Yaskawa INFORM job: plata_tarpez_cylinder_program.JBI

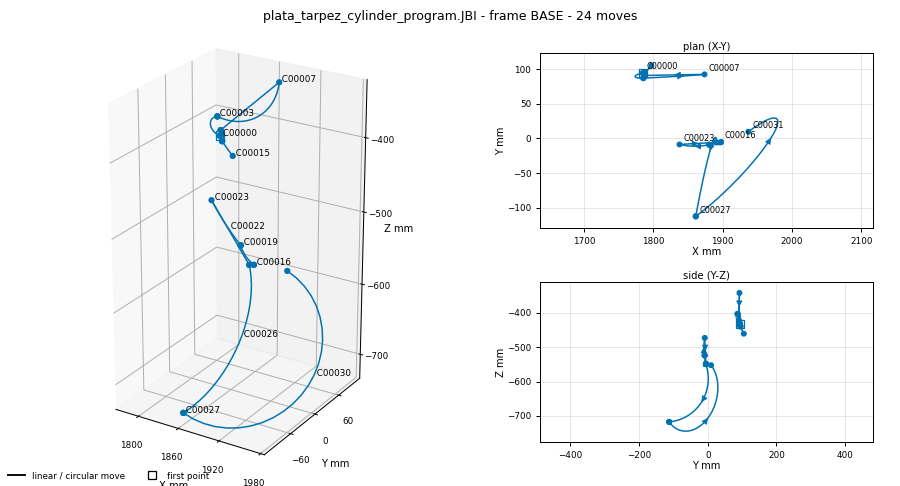
[picture p0: tool path of plata_tarpez_cylinder_program.JBI in frame BASE, 24 of 38 moves have a stored position in this frame; points joined in program order, loops and branches not executed]
/JOB
//NAME plata_tarpez_cylinder_program
//POS
///NPOS 32,0,32,0,0,0
///TOOL 0
///POSTYPE BASE
///RECTAN
///RCONF 0,0,0,0,0,0,0,0,0,0,0,0,0,0,0,0,0,0,0,0,0,0,0,0
C00000=1784.767004,94.191675,-431.505458,180.000000,-60.000000,6.127864
C00001=1784.767004,94.191675,-431.505458,180.000000,-60.000000,6.127864
C00002=1775.039434,88.021413,-411.039409,180.000000,-60.000000,7.554006
C00003=1785.526009,87.008169,-402.654234,-180.000000,-60.000000,8.255900
C00004=1785.526009,87.008169,-402.654234,-180.000000,-60.000000,8.255900
C00005=1785.526009,87.008169,-402.654234,-180.000000,-60.000000,8.255900
C00006=1813.588440,88.471809,-404.399549,-175.000000,-59.181249,9.143782
C00007=1873.697625,92.428351,-341.583881,175.000000,-33.351655,12.175617
C00008=1787.946995,90.909642,-422.120609,180.000000,-60.000000,6.802920
C00009=1787.946995,90.909642,-422.120609,180.000000,-60.000000,6.802920
C00010=1790.431356,93.825373,-431.135519,-180.000000,-60.000000,6.013660
C00011=1787.391263,95.251441,-438.765944,180.000000,-60.000000,5.494577
C00012=1787.391263,95.251441,-438.765944,180.000000,-60.000000,5.494577
C00013=1787.391263,95.251441,-438.765944,180.000000,-60.000000,5.494577
C00014=1790.708780,98.087857,-445.800605,-180.000000,-60.000000,4.731475
C00015=1797.176815,105.209463,-460.353029,180.000000,-60.000000,2.655850
C00016=1897.583937,-5.230695,-547.479957,180.000000,-60.000000,16.298157
C00017=1897.583937,-5.230695,-547.479957,180.000000,-60.000000,16.298157
C00018=1887.311406,-7.786471,-537.332214,-180.000000,-60.000000,15.451438
C00019=1880.512117,-8.938610,-523.580221,180.000000,-60.000000,14.334171
C00020=1880.512117,-8.938610,-523.580221,180.000000,-60.000000,14.334171
C00021=1880.512117,-8.938610,-523.580221,180.000000,-60.000000,14.334171
C00022=1863.998597,-11.006323,-503.995770,180.000000,-60.000000,12.058204
C00023=1837.651613,-8.596961,-472.556053,-180.000000,-60.000000,6.286549
C00024=1890.956692,-5.570875,-549.049019,-180.000000,-60.000000,16.288962
C00025=1890.956692,-5.570875,-549.049019,-180.000000,-60.000000,16.288962
C00026=1883.336474,-11.768567,-648.511835,180.000000,-60.000000,22.694763
C00027=1861.091301,-112.281106,-717.227974,180.000000,-60.000000,64.691502
C00028=1861.091301,-112.281106,-717.227974,180.000000,-60.000000,64.691502
C00029=1861.091301,-112.281106,-717.227974,180.000000,-60.000000,64.691502
C00030=1975.823049,11.866310,-688.422124,-180.000000,-60.000000,-170.270402
C00031=1936.915574,9.755960,-552.069704,180.000000,-60.000000,-159.283078
///POSTYPE PULSE
///PULSE
EX00000=0
EX00001=92160
EX00002=184320
EX00003=276480
///POSTYPE PULSE
///PULSE
EC00000=0
EC00001=0
EC00002=0
EC00003=0
EC00004=0
EC00005=0
EC00006=0
EC00007=0
EC00008=0
EC00009=0
EC00010=0
EC00011=0
EC00012=0
EC00013=0
EC00014=0
EC00015=0
EC00016=92160
EC00017=92160
EC00018=92160
EC00019=92160
EC00020=92160
EC00021=92160
EC00022=92160
EC00023=92160
EC00024=92160
EC00025=92160
EC00026=92160
EC00027=92160
EC00028=92160
EC00029=92160
EC00030=92160
EC00031=92160
//INST
///DATE 2023/08/07 13:53
///ATTR SC,RW,RJ
////FRAME BASE
///GROUP1 RB1,ST1
NOP
MOVJ P009 EX000 VJ=15.00
MOVJ P009 VJ=15.00
MOVJ C00000 EC00000 VJ=15.0
CALL JOB:SPYON
MOVC C00001 EC00001 V=150.0
MOVC C00002 EC00002 V=150.0
MOVC C00003 EC00003 V=150.0
MOVL C00004 EC00004 V=150.0
MOVC C00005 EC00005 V=150.0
MOVC C00006 EC00006 V=150.0
MOVC C00007 EC00007 V=150.0
MOVL C00008 EC00008 V=150.0
MOVC C00009 EC00009 V=150.0
MOVC C00010 EC00010 V=150.0
MOVC C00011 EC00011 V=150.0
MOVL C00012 EC00012 V=150.0
MOVC C00013 EC00013 V=150.0
MOVC C00014 EC00014 V=150.0
MOVC C00015 EC00015 V=150.0
CALL JOB:SPYOF
MOVJ P009 VJ=15.00
MOVJ C00016 EC00016 VJ=15.0
CALL JOB:SPYON
MOVC C00017 EC00017 V=150.0
MOVC C00018 EC00018 V=150.0
MOVC C00019 EC00019 V=150.0
MOVL C00020 EC00020 V=150.0
MOVC C00021 EC00021 V=150.0
MOVC C00022 EC00022 V=150.0
MOVC C00023 EC00023 V=150.0
MOVL C00024 EC00024 V=150.0
MOVC C00025 EC00025 V=150.0
MOVC C00026 EC00026 V=150.0
MOVC C00027 EC00027 V=150.0
MOVL C00028 EC00028 V=150.0
MOVC C00029 EC00029 V=150.0
MOVC C00030 EC00030 V=150.0
MOVC C00031 EC00031 V=150.0
CALL JOB:SPYOF
MOVJ P009 VJ=15.00
MOVJ P009 VJ=15.00
MOVJ P009 VJ=15.00
END
